Yaskawa INFORM job: USER_CART_S1_FLIP_UF3.JBI

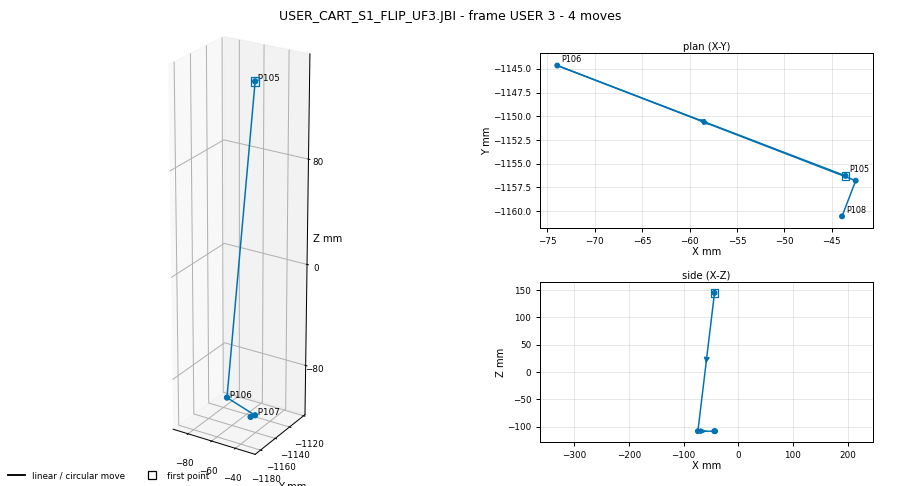
[picture p0: tool path of USER_CART_S1_FLIP_UF3.JBI in frame USER 3, 4 of 4 moves have a stored position in this frame; points joined in program order, loops and branches not executed]
/JOB
//NAME USER_CART_S1_FLIP_UF3
//POS
///NPOS 0,0,0,4,0,0
///TOOL 0
///USER 3
///POSTYPE USER
///RECTAN
///RCONF 1,0,0,0,0,0,0,0,0,0,0,0,0,0,0,0,0,0,0,0,0,0,0,0
P00105=-43.543,-1156.278,144.786,179.9929,0.0387,-21.0818
P00106=-73.955,-1144.635,-108.304,179.9901,0.0388,-21.0820
P00107=-42.467,-1156.784,-108.324,179.9891,0.0393,-21.0834
P00108=-43.911,-1160.550,-108.335,179.9891,0.0383,-21.0832
//INST
///DATE 2026/08/22 00:00
///ATTR SC,RW
///GROUP1 RB1
NOP
MOVJ P105 VJ=25.00
MOVL P106 V=150.0
MOVL P107 V=150.0
MOVL P108 V=150.0
END
